// TIA Portal V15.1 export
// export: Created 2026-01-15T16:29:49.1634389Z, ExportSetting WithDefaults, WithReadOnly, DisplayName Totally Integrated Automation Portal, DisplayVersion V15.1 Update 8, DisplayName TIA Portal Openness, DisplayVersion V15.1 Update 8, DisplayName STEP 7 Professional, DisplayVersion V15.1 Update 8, DisplayName WinCC Advanced, DisplayVersion V15.1 Update 8
VAR_GLOBAL   // PLC tag table "In_Put"
   "I_TH. NOI TRON" AT %I0.0 : Bool;   // Input_Tín hiệu nồi trộn
   "I_TH. BTX" AT %I0.1 : Bool;   // Input_Tín hiệu băng tải xiên
   "I_TH. BTN" AT %I0.2 : Bool;   // Input_Tín hiệu băng tải ngang
   "I_TH. TANG SAY" AT %I0.3 : Bool;   // Input_Tín hiệu tang sấy cốt liệu
   "I_TH. GAU COT LIEU" AT %I0.4 : Bool;   // Input_Tín hiệu gàu tải cốt liệu nóng
   "I_TH. GAU F/D" AT %I0.5 : Bool;   // Input_Tín hiệu gàu tải phụ gia bột
   "I_TH. SANG RUNG" AT %I0.6 : Bool;   // Input_Tín hiệu sàng rung cốt liệu nóng
   "I_TH. CUA DONG" AT %I0.7 : Bool;   // Input_Tín hiệu cửa nồi trộn đóng
   "I_TH. CUA MO" AT %I1.0 : Bool;   // Input_Tín hiệu cửa nồi trộn mở
   "I_TH. MNK" AT %I1.1 : Bool;   // Input_Tín hiệu máy nén khí chạy
   "I_TH. TRAN AG1" AT %I1.2 : Bool;   // Input_Tín hiệu báo tràn silo AG1
   "I_TH. TRAN AG2" AT %I1.3 : Bool;   // Input_Tín hiệu báo tràn silo AG2
   "I_TH. TRAN AG3" AT %I1.4 : Bool;   // Input_Tín hiệu báo tràn silo AG3
   "I_TH. TRAN AG4" AT %I1.5 : Bool;   // Input_Tín hiệu báo tràn silo AG4
   "I_TH. TRAN AG5" AT %I2.0 : Bool;   // Input_Tín hiệu báo tràn silo AG5
   "I_TH. TRAN FD1" AT %I2.1 : Bool;   // Input_Tín hiệu báo tràn silo F/D
   "I_TH. TRAN SB1" AT %I2.2 : Bool;   // Input_Tín hiệu báo tràn silo SBS
   "I_TH. SILO FD HIGHT" AT %I2.3 : Bool;   // Input_Tín hiệu báo mức cao silo chứa F/D
   "I_TH. SILO FD LOW" AT %I2.4 : Bool;   // Input_Tín hiệu báo mức thấp silo chứa F/D
   "TH. NOI TRON" AT %M400.0 : Bool;   // Tín hiệu nồi trộn
   "TH. BTX" AT %M400.1 : Bool;   // Tín hiệu băng tải xiên
   "TH. BTN" AT %M400.2 : Bool;   // Tín hiệu băng tải ngang
   "TH. TANG SAY" AT %M400.3 : Bool;   // Tín hiệu tang sấy cốt liệu
   "TH. GAU COT LIEU" AT %M400.4 : Bool;   // Tín hiệu gàu tải cốt liệu nóng
   "TH. GAU F/D" AT %M400.5 : Bool;   // Tín hiệu gàu tải phụ gia bột
   "TH. SANG RUNG" AT %M400.6 : Bool;   // Tín hiệu sàng rung cốt liệu nóng
   "TH. CUA DONG" AT %M400.7 : Bool;   // Tín hiệu cửa nồi trộn đóng
   "TH. CUA MO" AT %M401.0 : Bool;   // Tín hiệu cửa nồi trộn mở
   "TH. MNK" AT %M401.1 : Bool;   // Tín hiệu máy nén khí chạy
   "TH. TRAN AG1" AT %M401.2 : Bool;   // Tín hiệu báo tràn silo AG1
   "TH. TRAN AG2" AT %M401.3 : Bool;   // Tín hiệu báo tràn silo AG2
   "TH. TRAN AG3" AT %M401.4 : Bool;   // Tín hiệu báo tràn silo AG3
   "TH. TRAN AG4" AT %M401.5 : Bool;   // Tín hiệu báo tràn silo AG4
   "TH. TRAN AG5" AT %M401.6 : Bool;   // Tín hiệu báo tràn silo AG5
   "TH. TRAN FD1" AT %M401.7 : Bool;   // Tín hiệu báo tràn silo F/D
   "TH. TRAN SB1" AT %M402.0 : Bool;   // Tín hiệu báo tràn silo SBS
   "TH. SILO FD HIGHT" AT %M402.1 : Bool;   // Tín hiệu báo mức cao silo chứa F/D
   "TH. SILO FD LOW" AT %M402.2 : Bool;   // Tín hiệu báo mức thấp silo chứa F/D
   "TH_CNM SIM" AT %M402.3 : Bool;
   "TH_CND SIM" AT %M402.4 : Bool;
END_VAR
